Omron CX-Programmer project NewProject (CX-Programmer 9.75)

# PLC NewPLC1: CP1L-E EM

## Global symbols (name address type ; comment)
0.00 BOOL  ; Emergency
100.00 BOOL  ; KM1
100.01 BOOL  ; KM2
100.02 BOOL  ; KM3
100.03 BOOL  ; KM4
100.04 BOOL  ; KM5A
100.05 BOOL  ; KM5B
100.06 BOOL  ; KM6A
100.07 BOOL  ; KM6B
101.00 BOOL  ; Sarin
20.00 BOOL  ; EMG OK
20.01 BOOL  ; OK Start Belts
30.00 BOOL  ; Start Load 5
30.01 BOOL  ; Start Load 6
30.02 BOOL  ; Start Load 7
30.03 BOOL  ; stop 4
30.04 BOOL  ; stop 5
40.00 BOOL  ; Start Belts
50.00 BOOL  ; Stop Cycle
60.00 BOOL  ; ALARM
D100 CHANNEL  ; Silo 5 Level Time
D101 CHANNEL  ; Time Level 6
D102 CHANNEL  ; Time Level 7
T0000 BOOL  ; Time Level 5
T0001 BOOL  ; Time To Start Belts 5
T0002 BOOL  ; Level 6 Time
T0003 BOOL  ; Time To Start Belts 6
T0004 BOOL  ; Level 7 Time
T0005 BOOL  ; Time To Start Belts 7
W0.00 BOOL  ; EMG
W0.01 BOOL  ; Level 5 ON
W0.02 BOOL  ; Level 6
W0.03 BOOL  ; Level 7
W0.04 BOOL  ; OverLoad Trip
W10.00 BOOL  ; MM5A
W10.01 BOOL  ; MM6A
W10.02 BOOL  ; MM4
W10.03 BOOL  ; MM3
W10.04 BOOL  ; MM2
W10.05 BOOL  ; MM1
W10.06 BOOL  ; MM6B
W10.07 BOOL  ; MM5B
W1.00 BOOL  ; M1
W1.01 BOOL  ; M2
W1.02 BOOL  ; M3
W1.03 BOOL  ; M4
W1.04 BOOL  ; M5A
W1.05 BOOL  ; M5B
W1.06 BOOL  ; M6A
W1.07 BOOL  ; M6B
W1.08 BOOL  ; Sarin+Fanar
W2.00 BOOL  ; Start Load 6
W2.01 BOOL  ; Start  Load 7
W5.00 BOOL  ; Stop M1
W5.01 BOOL  ; STOP M2
W5.02 BOOL  ; STOP M3
W5.03 BOOL  ; STOP M4
W5.04 BOOL  ; STOP M5
W5.05 BOOL  ; STOP M6
W6.10 BOOL  ; Level 5 Off
W6.11 BOOL  ; Level 6 Off
W6.12 BOOL  ; Level 7 Off

## Program New_Program (cyclic task 0)

### Section I_O

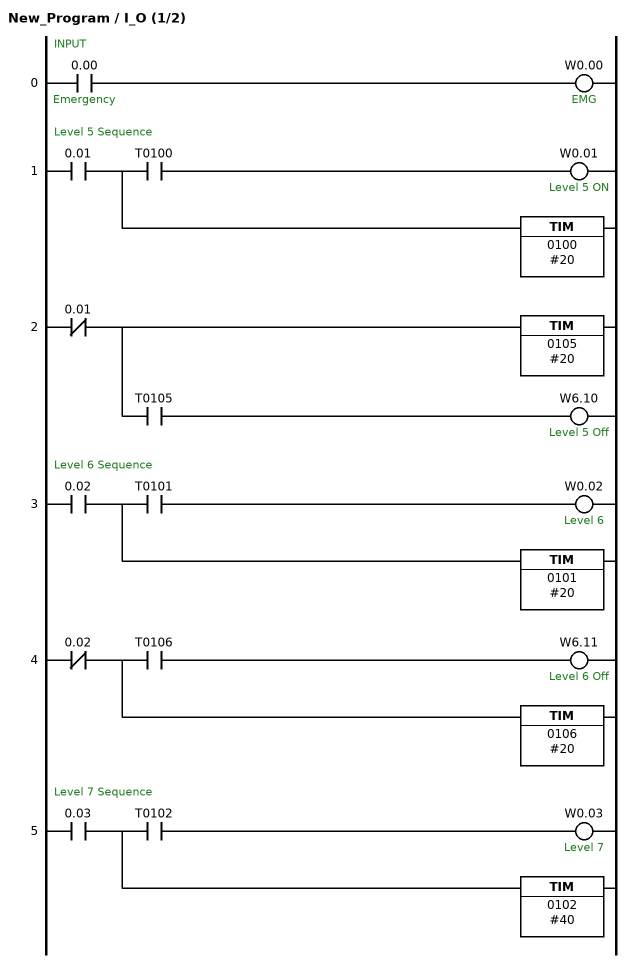
; rung 0: INPUT
LD 0.00  ; Emergency
OUT W0.00  ; EMG
; rung 1: Level 5 Sequence
LD 0.01
OUT TR0
AND T0100
OUT W0.01  ; Level 5 ON
LD TR0
TIM 0100 #20
; rung 2
LDNOT 0.01
TIM 0105 #20
AND T0105
OUT W6.10  ; Level 5 Off
; rung 3: Level 6 Sequence
LD 0.02
OUT TR0
AND T0101
OUT W0.02  ; Level 6
LD TR0
TIM 0101 #20
; rung 4
LDNOT 0.02
OUT TR0
AND T0106
OUT W6.11  ; Level 6 Off
LD TR0
TIM 0106 #20
; rung 5: Level 7 Sequence
LD 0.03
OUT TR0
AND T0102
OUT W0.03  ; Level 7
LD TR0
TIM 0102 #40

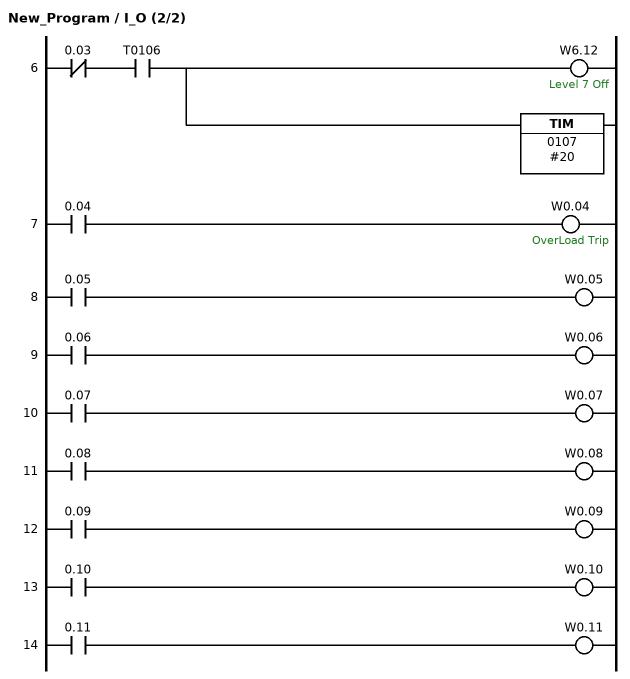
; rung 6
LDNOT 0.03
AND T0106
OUT W6.12  ; Level 7 Off
TIM 0107 #20
; rung 7
LD 0.04
OUT W0.04  ; OverLoad Trip
; rung 8
LD 0.05
OUT W0.05
; rung 9
LD 0.06
OUT W0.06
; rung 10
LD 0.07
OUT W0.07
; rung 11
LD 0.08
OUT W0.08
; rung 12
LD 0.09
OUT W0.09
; rung 13
LD 0.10
OUT W0.10
; rung 14
LD 0.11
OUT W0.11

### Section Main

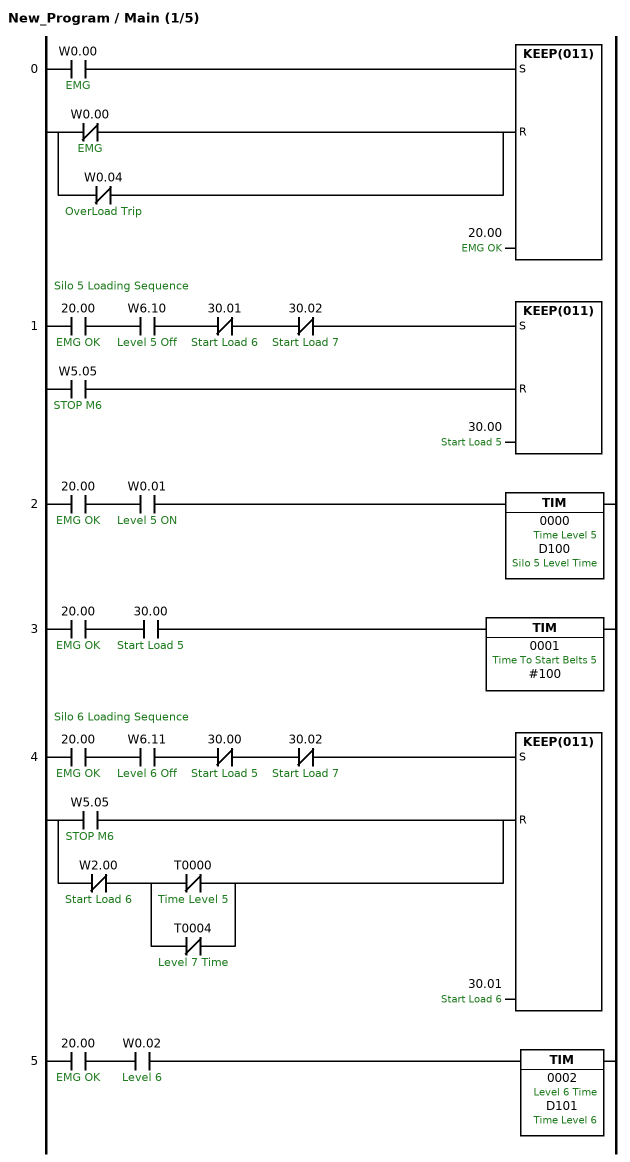
; rung 0
LD W0.00  ; EMG
LDNOT W0.00  ; EMG
ORNOT W0.04  ; OverLoad Trip
KEEP(011) 20.00  ; EMG OK
; rung 1: Silo 5 Loading Sequence
LD 20.00  ; EMG OK
AND W6.10  ; Level 5 Off
ANDNOT 30.01  ; Start Load 6
ANDNOT 30.02  ; Start Load 7
LD W5.05  ; STOP M6
KEEP(011) 30.00  ; Start Load 5
; rung 2
LD 20.00  ; EMG OK
AND W0.01  ; Level 5 ON
TIM 0000 D100  ; Silo 5 Level Time, Time Level 5
; rung 3
LD 20.00  ; EMG OK
AND 30.00  ; Start Load 5
TIM 0001 #100  ; Time To Start Belts 5
; rung 4: Silo 6 Loading Sequence
LD 20.00  ; EMG OK
AND W6.11  ; Level 6 Off
ANDNOT 30.00  ; Start Load 5
ANDNOT 30.02  ; Start Load 7
LD W5.05  ; STOP M6
LDNOT W2.00  ; Start Load 6
LDNOT T0000  ; Time Level 5
ORNOT T0004  ; Level 7 Time
ANDLD
ORLD
KEEP(011) 30.01  ; Start Load 6
; rung 5
LD 20.00  ; EMG OK
AND W0.02  ; Level 6
TIM 0002 D101  ; Time Level 6, Level 6 Time

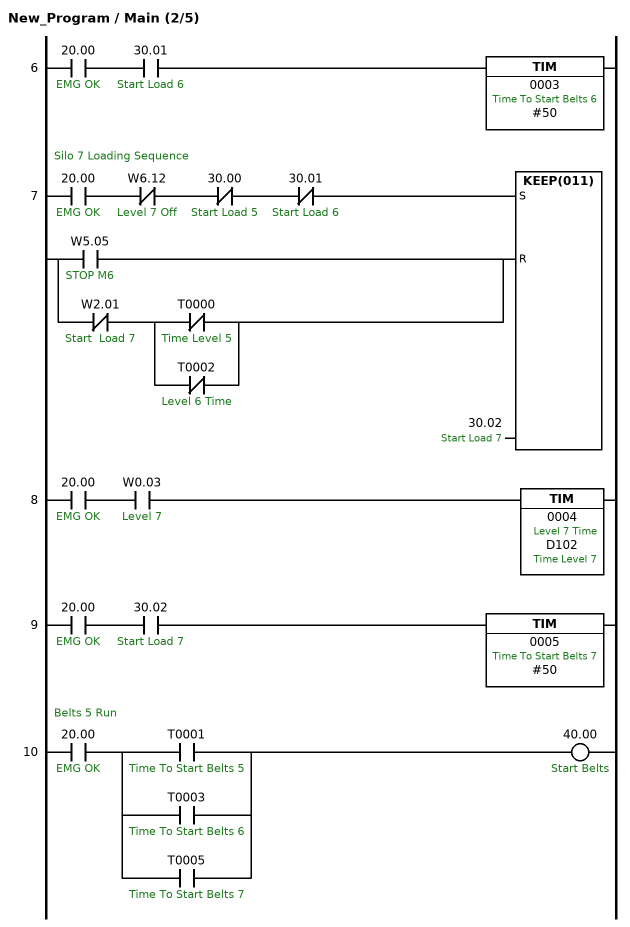
; rung 6
LD 20.00  ; EMG OK
AND 30.01  ; Start Load 6
TIM 0003 #50  ; Time To Start Belts 6
; rung 7: Silo 7 Loading Sequence
LD 20.00  ; EMG OK
ANDNOT W6.12  ; Level 7 Off
ANDNOT 30.00  ; Start Load 5
ANDNOT 30.01  ; Start Load 6
LD W5.05  ; STOP M6
LDNOT W2.01  ; Start  Load 7
LDNOT T0000  ; Time Level 5
ORNOT T0002  ; Level 6 Time
ANDLD
ORLD
KEEP(011) 30.02  ; Start Load 7
; rung 8
LD 20.00  ; EMG OK
AND W0.03  ; Level 7
TIM 0004 D102  ; Time Level 7, Level 7 Time
; rung 9
LD 20.00  ; EMG OK
AND 30.02  ; Start Load 7
TIM 0005 #50  ; Time To Start Belts 7
; rung 10: Belts 5 Run
LD 20.00  ; EMG OK
LD T0001  ; Time To Start Belts 5
OR T0003  ; Time To Start Belts 6
OR T0005  ; Time To Start Belts 7
ANDLD
OUT 40.00  ; Start Belts

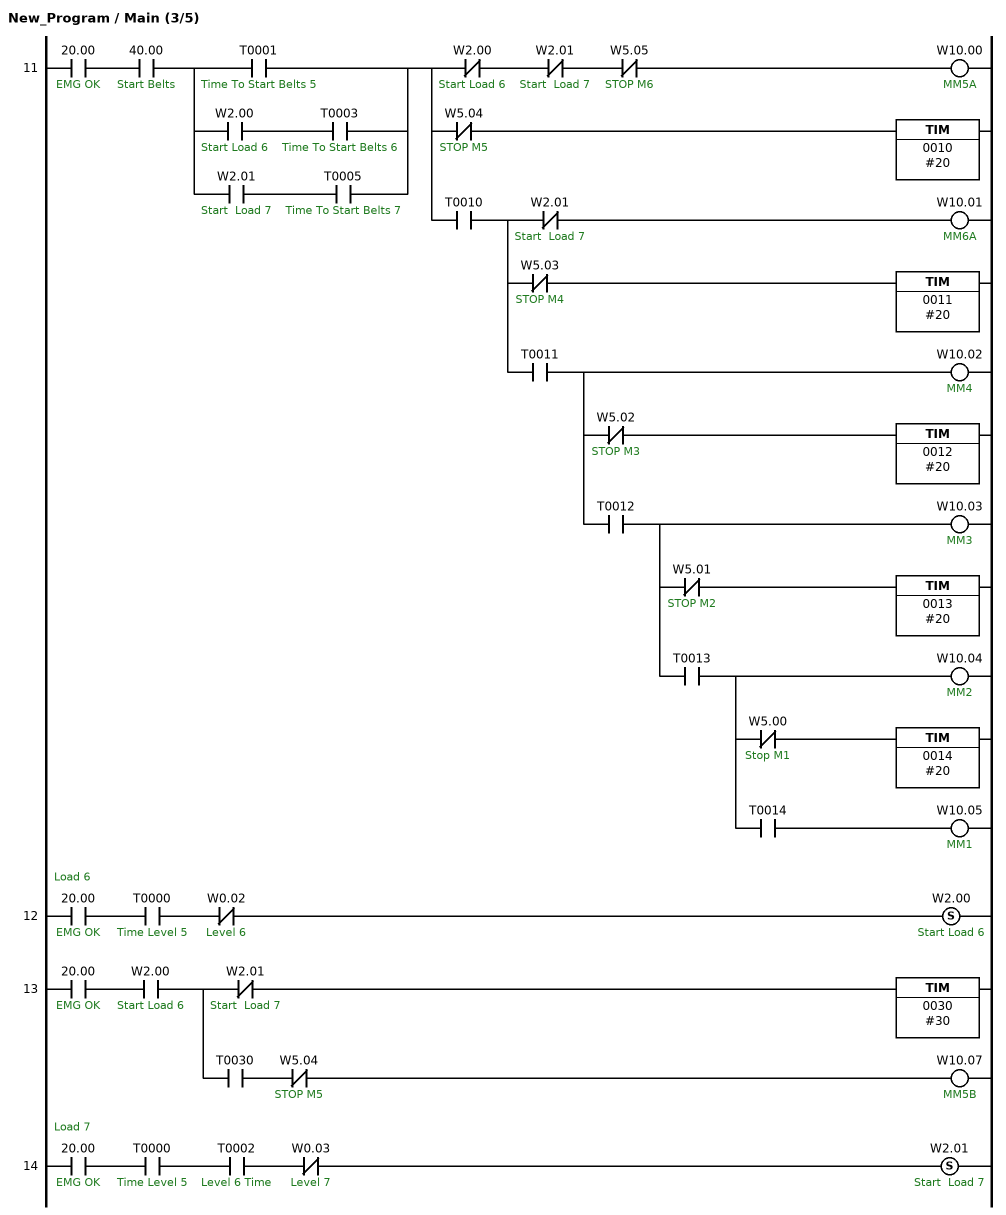
; rung 11
LD 20.00  ; EMG OK
AND 40.00  ; Start Belts
LD T0001  ; Time To Start Belts 5
LD W2.00  ; Start Load 6
AND T0003  ; Time To Start Belts 6
ORLD
LD W2.01  ; Start  Load 7
AND T0005  ; Time To Start Belts 7
ORLD
ANDLD
OUT TR0
ANDNOT W2.00  ; Start Load 6
ANDNOT W2.01  ; Start  Load 7
ANDNOT W5.05  ; STOP M6
OUT W10.00  ; MM5A
LD TR0
ANDNOT W5.04  ; STOP M5
TIM 0010 #20
LD TR0
AND T0010
OUT TR0
ANDNOT W2.01  ; Start  Load 7
OUT W10.01  ; MM6A
LD TR0
ANDNOT W5.03  ; STOP M4
TIM 0011 #20
LD TR0
AND T0011
OUT TR0
OUT W10.02  ; MM4
ANDNOT W5.02  ; STOP M3
TIM 0012 #20
LD TR0
AND T0012
OUT TR0
OUT W10.03  ; MM3
ANDNOT W5.01  ; STOP M2
TIM 0013 #20
LD TR0
AND T0013
OUT TR0
OUT W10.04  ; MM2
ANDNOT W5.00  ; Stop M1
TIM 0014 #20
LD TR0
AND T0014
OUT W10.05  ; MM1
; rung 12: Load 6
LD 20.00  ; EMG OK
AND T0000  ; Time Level 5
ANDNOT W0.02  ; Level 6
SET W2.00  ; Start Load 6
; rung 13
LD 20.00  ; EMG OK
AND W2.00  ; Start Load 6
OUT TR0
ANDNOT W2.01  ; Start  Load 7
TIM 0030 #30
LD TR0
AND T0030
ANDNOT W5.04  ; STOP M5
OUT W10.07  ; MM5B
; rung 14: Load 7
LD 20.00  ; EMG OK
AND T0000  ; Time Level 5
AND T0002  ; Level 6 Time
ANDNOT W0.03  ; Level 7
SET W2.01  ; Start  Load 7

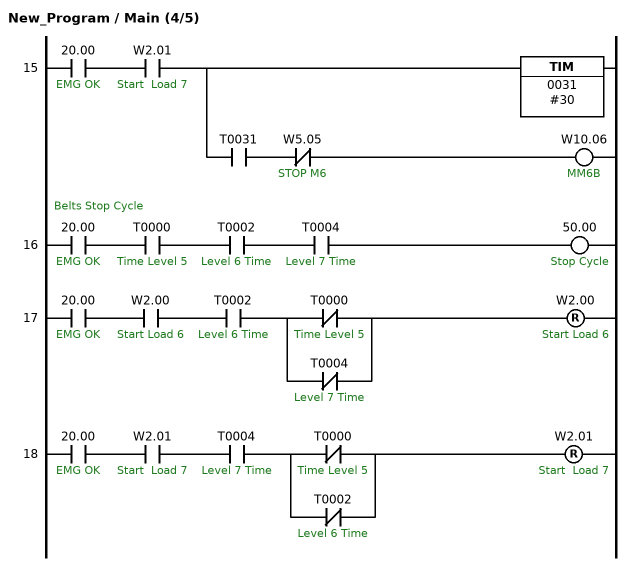
; rung 15
LD 20.00  ; EMG OK
AND W2.01  ; Start  Load 7
TIM 0031 #30
AND T0031
ANDNOT W5.05  ; STOP M6
OUT W10.06  ; MM6B
; rung 16: Belts Stop Cycle
LD 20.00  ; EMG OK
AND T0000  ; Time Level 5
AND T0002  ; Level 6 Time
AND T0004  ; Level 7 Time
OUT 50.00  ; Stop Cycle
; rung 17
LD 20.00  ; EMG OK
AND W2.00  ; Start Load 6
AND T0002  ; Level 6 Time
LDNOT T0000  ; Time Level 5
ORNOT T0004  ; Level 7 Time
ANDLD
RSET W2.00  ; Start Load 6
; rung 18
LD 20.00  ; EMG OK
AND W2.01  ; Start  Load 7
AND T0004  ; Level 7 Time
LDNOT T0000  ; Time Level 5
ORNOT T0002  ; Level 6 Time
ANDLD
RSET W2.01  ; Start  Load 7

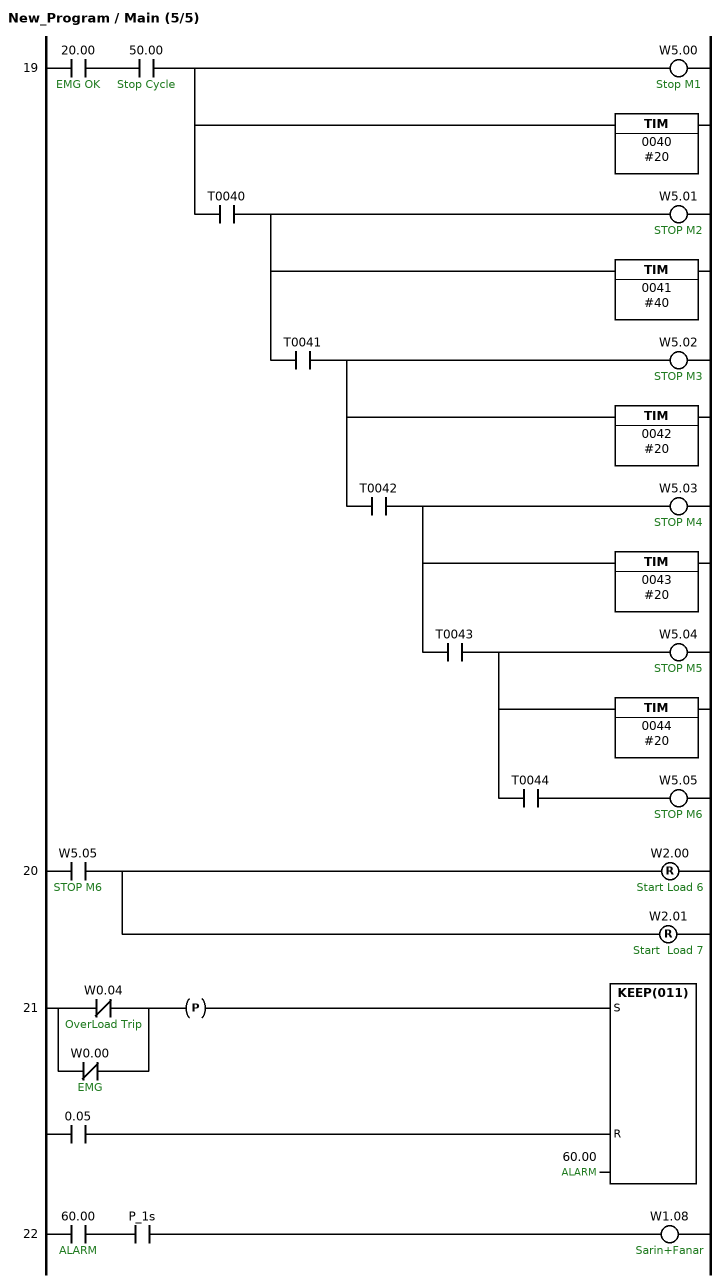
; rung 19
LD 20.00  ; EMG OK
AND 50.00  ; Stop Cycle
OUT W5.00  ; Stop M1
TIM 0040 #20
AND T0040
OUT W5.01  ; STOP M2
TIM 0041 #40
AND T0041
OUT W5.02  ; STOP M3
TIM 0042 #20
AND T0042
OUT W5.03  ; STOP M4
TIM 0043 #20
AND T0043
OUT W5.04  ; STOP M5
TIM 0044 #20
AND T0044
OUT W5.05  ; STOP M6
; rung 20
LD W5.05  ; STOP M6
RSET W2.00  ; Start Load 6
RSET W2.01  ; Start  Load 7
; rung 21
LDNOT W0.04  ; OverLoad Trip
ORNOT W0.00  ; EMG
UP(521)
LD 0.05
KEEP(011) 60.00  ; ALARM
; rung 22
LD 60.00  ; ALARM
AND P_1s
OUT W1.08  ; Sarin+Fanar

### Section Outputs

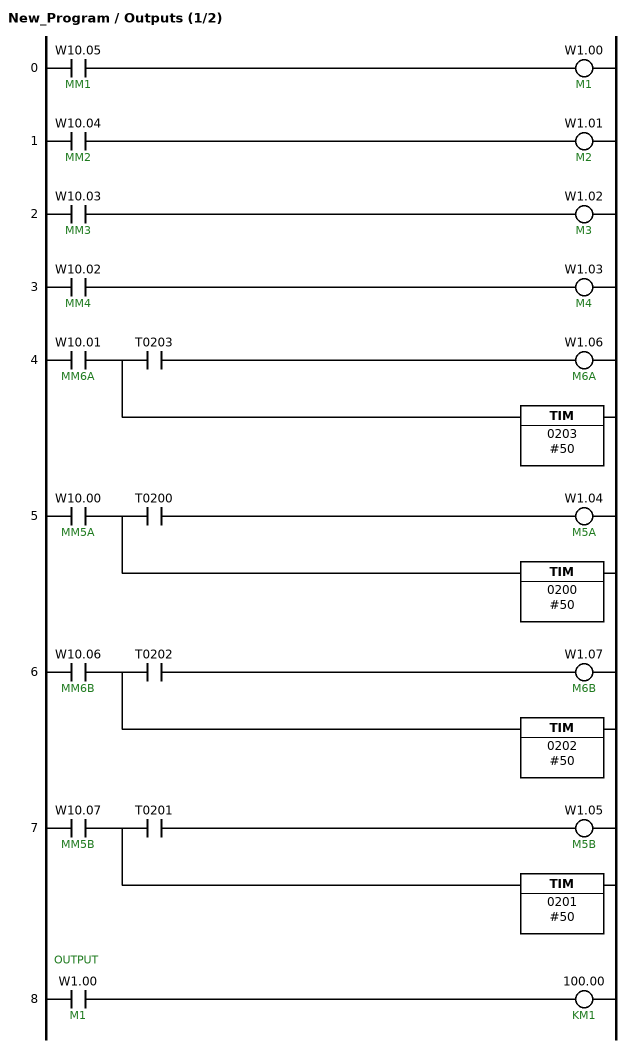
; rung 0
LD W10.05  ; MM1
OUT W1.00  ; M1
; rung 1
LD W10.04  ; MM2
OUT W1.01  ; M2
; rung 2
LD W10.03  ; MM3
OUT W1.02  ; M3
; rung 3
LD W10.02  ; MM4
OUT W1.03  ; M4
; rung 4
LD W10.01  ; MM6A
OUT TR0
AND T0203
OUT W1.06  ; M6A
LD TR0
TIM 0203 #50
; rung 5
LD W10.00  ; MM5A
OUT TR0
AND T0200
OUT W1.04  ; M5A
LD TR0
TIM 0200 #50
; rung 6
LD W10.06  ; MM6B
OUT TR0
AND T0202
OUT W1.07  ; M6B
LD TR0
TIM 0202 #50
; rung 7
LD W10.07  ; MM5B
OUT TR0
AND T0201
OUT W1.05  ; M5B
LD TR0
TIM 0201 #50
; rung 8: OUTPUT
LD W1.00  ; M1
OUT 100.00  ; KM1

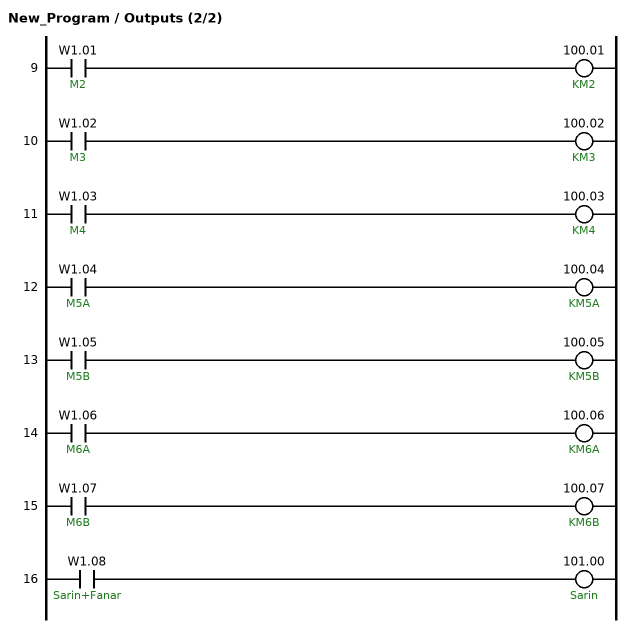
; rung 9
LD W1.01  ; M2
OUT 100.01  ; KM2
; rung 10
LD W1.02  ; M3
OUT 100.02  ; KM3
; rung 11
LD W1.03  ; M4
OUT 100.03  ; KM4
; rung 12
LD W1.04  ; M5A
OUT 100.04  ; KM5A
; rung 13
LD W1.05  ; M5B
OUT 100.05  ; KM5B
; rung 14
LD W1.06  ; M6A
OUT 100.06  ; KM6A
; rung 15
LD W1.07  ; M6B
OUT 100.07  ; KM6B
; rung 16
LD W1.08  ; Sarin+Fanar
OUT 101.00  ; Sarin

### Section END
; rung 0
END(001)